(* IEC 61131-3 sources: teller/JD_Teller_LC2_V11/Class/ActScreenWindow, 1 file *)

(* ---- ActScreenWindow.st ---- *)
(*!
<Class
	Name               = "ActScreenWindow"
	Revision           = "0.0"
	RealtimeTask       = "false"
	CyclicTask         = "false"
	BackgroundTask     = "false"
	Sigmatek           = "false"
	OSInterface        = "false"
	HighPriority       = "false"
	Automatic          = "false"
	UpdateMode         = "Prescan"
	SharedCommandTable = "true"
	Objectsize         = "(410,120)">
	<Channels>
		<Server Name="ActScreenNr" Visualized="true" Initialize="false" WriteProtected="true" Retentive="false"/>
		<Server Name="ActWindowNr" Visualized="true" Initialize="false" WriteProtected="true" Retentive="false"/>
	</Channels>
	<Network Name="ActScreenWindow">
		<!-- List of Components in this network -->
		<Components>
			<Object
				Name       = "_base"
				Class      = "_Global"
				Position   = "(218,120)"
				Visualized = "false">
				<Channels>
					<Server Name="Server0"/>
					<Client Name="Lse"/>
				</Channels>
			</Object>
		</Components>
		<Comments>
		</Comments>
		<!-- List of Connections in this network -->
		<Connections>
			<Connection Source="this.Server0" Destination="_base.Server0" Vertices="(690,210),(518,210),"/>
			<Connection Source="_base.Lse" Destination="this.Lse" Vertices="(218,210),(38,210),"/>
		</Connections>
		<!-- Headerfiles -->
		<Options>
		</Options>
	</Network>
</Class>
*)
#pragma using _Global

ActScreenWindow : CLASS
: _Global
  //Servers:
	ActScreenNr 	: SvrCh_DINT;
	ActWindowNr 	: SvrCh_DINT;
  //Clients:
  //Variables:
  //Functions:

	FUNCTION VIRTUAL GLOBAL IF_WindowRun
		VAR_INPUT
			whoami 	: ^_WHOAMI;
			pic 	: ^void;
			event 	: ^_EVENT;
		END_VAR;
  //Tables:
	FUNCTION @STD
		VAR_OUTPUT
			ret_code	: CONFSTATES;
		END_VAR;
	FUNCTION GLOBAL TAB @CT_;
END_CLASS;

FUNCTION VIRTUAL GLOBAL ActScreenWindow::IF_WindowRun
	VAR_INPUT
		whoami 	: ^_WHOAMI;
		pic 	: ^void;
		event 	: ^_EVENT;
	END_VAR

	case whoami^.ima of

	IMA_PICTURE:
		ActScreenNr := to_dint whoami^.no;

	IMA_WINDOW:
		ActWindowNr := to_dint whoami^.no;
	end_case;

END_FUNCTION
